// Provide logging 
FUNCTION_BLOCK FB_Logger IMPLEMENTS I_Logger
VAR_INPUT
	eLogLevel:				E_LogLevel:= E_LogLevel.Verbose;
END_VAR
VAR_OUTPUT
    bInfo:					BOOL;
    bWarning:				BOOL;
    bError:					BOOL;
    bCritical:				BOOL;
END_VAR
VAR
	aMessages:				ARRAY[0..99] OF FB_Message; // Message store
    nMessages:				UINT := 0;                     // Message count
	{attribute 'hide'} 
	nIndex: 				UINT;
	nTimestamp:				LINT;
END_VAR

// clean up after 1 secound
IF nTimestamp < TwinCAT_SystemInfoVarList._TaskInfo[GETCURTASKINDEXEX()].DcTaskTime THEN // 1 second = 1e9 ns
	nTimestamp := TwinCAT_SystemInfoVarList._TaskInfo[GETCURTASKINDEXEX()].DcTaskTime + 1000000000;
	nIndex := 0;
	WHILE nIndex < nMessages DO
		IF aMessages[nIndex].bActive THEN
			aMessages[nIndex].bActive:= FALSE;
			nIndex := nIndex + 1;
		ELSE
			MEMMOVE(ADR(aMessages[nIndex]), ADR(aMessages[nIndex + 1]), SIZEOF(ST_Message) * (nMessages - nIndex));
			nMessages := nMessages - 1;
			bInfo:=	FALSE;
			bWarning:=	FALSE;
			bError:= FALSE;
			bCritical:= FALSE;
		END_IF
	END_WHILE
END_IF

METHOD PUBLIC M_Log : BOOL
VAR_INPUT
	fbMessage:			FB_Message;
END_VAR
VAR
END_VAR
IF eLogLevel > fbMessage.eLogLevel THEN
	M_Log:= TRUE;
	RETURN;
END_IF

CASE fbMessage.eLogLevel OF
	E_LogLevel.Info:
    	bInfo:= TRUE;
		
	E_LogLevel.Warning:		
    	bWarning:= TRUE;
		
	E_LogLevel.Error:
    	bError:= TRUE;
		
	E_LogLevel.Critical:
    	bCritical:= TRUE;
		
	ELSE
		;
END_CASE


// Find
FOR nIndex := 0 TO nMessages DO
    IF aMessages[nIndex].sMessage = fbMessage.sMessage AND_THEN aMessages[nIndex].sSource = fbMessage.sSource THEN
        aMessages[nIndex].bActive:= TRUE;
		M_Log := TRUE;
        RETURN;
    END_IF
END_FOR

// else Add
IF nMessages < 99 THEN
	nIndex := nMessages;
	fbMessage.bActive:= TRUE;
    aMessages[nMessages]:= fbMessage;;
    nMessages := nMessages + 1;
	M_Log := TRUE;
END_IF
END_METHOD

PROPERTY PUBLIC P_LogLevel : E_LogLevel
GET
P_LogLevel:= eLogLevel;
END_GET
SET
eLogLevel:= P_LogLevel;
END_SET
END_PROPERTY

END_FUNCTION_BLOCK

(* stored: Version 1.1.0.1
   POU FB_Logger: Id {65f70f38-14b4-40c0-9ff9-f567428dadcd}, SpecialFunc None
   Method M_Log: Id {c925afc5-8e57-47da-84bb-210c829a3dd4}
   Property P_LogLevel: Id {1c739022-3d6f-4ecb-abf9-2f9944cdc386}
   Get Get: Id {92f636fd-e8a2-488e-a20a-d9bd7d8e0a21}
   Set Set: Id {98e4e2b1-517c-43c2-870d-a5a57ae02ec1} *)
